// TIA Portal project "TestingMurr" (V18)

(* hardware
DEVICE "S7-1200 station_1"  S7-1200 Station
   slot 0: "Rack_0"  S7-1200 Rack  Rack  V1.0
   slot 1: "PLC_1"  CPU 1212FC DC/DC/DC  6ES7 212-1AF40-0XB0  V4.6
DEVICE "GSD device_1"  GSD.Device.PN
   slot 0: "Rack"  Rack  V1.0
   slot 0: "IMPACT67-Pro"  54630 IMPACT67 Pro PNIO DIO8 IOL8 M12L 5P  54630  V1.5.0
      slot 0: "54630 IMPACT67 Pro PNIO DIO8 IOL8 M12L 5P_1"  54630 IMPACT67 Pro PNIO DIO8 IOL8 M12L 5P
      slot 1: "54630 IMPACT67 Pro PNIO DIO8 IOL8 M12L 5P"  54630 IMPACT67 Pro PNIO DIO8 IOL8 M12L 5P
         slot 1: "Port 1"  Port 1
         slot 2: "Port 2"  Port 2
      slot 1: "IMPACT67 Pro device_1"  IMPACT67 Pro device
         slot 0: "SIO data / Module parameters"  SIO data / Module parameters
      slot 2: "IMPACT67 Pro options_1"  IMPACT67 Pro options
   slot 1: "PortX0-59719 MVP12-P6 DIO16 8xM12A IOLA12 B0"  59719 MVP12-P6 DIO16 8xM12A IOLA12 B0
   slot 2: "Standard digital input"  Standard digital input
   slot 3: "Deactivated_1"  Deactivated
   slot 4: "PortX3-500x-00501-1300001 IOL AI-U/I-STR-MULT-PAR"  500x-00501-1300001 IOL AI-U/I-STR-MULT-PAR
   slot 5: "PortX4-Contrinex _IDWE-M12MM-NMS-A0"  IO-Link In/Out 04/02 bytes + PQI
   slot 6: "Web server"  Web server
   slot 6: "Standard digital output"  Standard digital output
   slot 7: "PortX6-OMRON_E3AS_HL500LMN"  IO-Link In/Out 04/02 bytes + PQI
   slot 8: "PortX7-TURCK_BN1F360V_QR20-IOLX3-H1141"  IO-Link In/Out 08/02 bytes + PQI
*)

// ===== PLC "PLC_1"  CPU 1212FC DC/DC/DC =====

VAR_GLOBAL   // PLC tag table "Default tag table"
   "iwMurrIOLINKData_SIO_IN" AT %I100.0 : "DUT_Murr_Submodule 1_SIO_PortBase_Pin";
   "iwMurrIOLINKData_X4_IN" AT %I114.0 : "DUT_RawArray_Length4";   // PortX4-Contrinex _IDWE-M12MM-NMS-A0
   "iwMurrIOLINKData_X6_IN" AT %I120.0 : "DUT_RawArray_Length4";   // PortX6-OMRON_E3AS_HL500LMN
   "iwMurrIOLINKData_X3_IN" AT %I110.0 : "DUT_RawArray_Length2";   // PortX3-500x-00501-1300001 IOL AI-U/I-STR-MULT-PAR
   "iwMurrIOLINKData_X3_IN_PQI" AT %IB112 : Byte;
   "iwMurrIOLINKData_X4_IN_PQI" AT %IB118 : Byte;
   "iwMurrIOLINKData_IN_X6_PQI" AT %IB124 : Byte;
   "iwMurrIOLINKData_X0_IN" AT %I102.0 : "DUT_RawArray_Length4";   // PortX0-59719 MVP12-P6 DIO16 8xM12A IOLA12 B0
   "iwMurrIOLINKData_X7_IN" AT %I126.0 : "DUT_RawArray_Length8";   // PortX7-TURCK_BN1F360V_QR20-IOLX3-H1141
   "iwMurrIOLINKData_X7_IN_PQI" AT %IB134 : Byte;
   "iwMurrIOLINKData_X0_OUT" AT %Q102.0 : "DUT_RawArray_Length2";
   "iwMurrIOLINKData_SIO_OUT" AT %Q100.0 : "DUT_Murr_Submodule 1_SIO_PortBase_Pin";
   "iwMurrIOLINKData_X5_IN_PQI" AT %IB138 : Byte;   // PortX7-TURCK_BN1F360V_QR20-IOLX3-H1141
   "System_Byte" AT %MB1 : Byte;
   "FirstScan" AT %M1.0 : Bool;
   "DiagStatusUpdate" AT %M1.1 : Bool;
   "AlwaysTRUE" AT %M1.2 : Bool;
   "AlwaysFALSE" AT %M1.3 : Bool;
   "Clock_Byte" AT %MB0 : Byte;
   "Clock_10Hz" AT %M0.0 : Bool;
   "Clock_5Hz" AT %M0.1 : Bool;
   "Clock_2.5Hz" AT %M0.2 : Bool;
   "Clock_2Hz" AT %M0.3 : Bool;
   "Clock_1.25Hz" AT %M0.4 : Bool;
   "Clock_1Hz" AT %M0.5 : Bool;
   "Clock_0.625Hz" AT %M0.6 : Bool;
   "Clock_0.5Hz" AT %M0.7 : Bool;
END_VAR

TYPE "DUT_Murr_Submodule 1_SIO_PortBase_Pin"
   STRUCT
      PortX0Pin4 : Bool;
      PortX0Pin2 : Bool;
      PortX1Pin4 : Bool;
      PortX1Pin2 : Bool;
      PortX2Pin4 : Bool;
      PortX2Pin2 : Bool;
      PortX3Pin4 : Bool;
      PortX3Pin2 : Bool;
      PortX4Pin4 : Bool := false;
      PortX4Pin2 : Bool := false;
      PortX5Pin4 : Bool := false;
      PortX5Pin2 : Bool := false;
      PortX6Pin4 : Bool := false;
      PortX6Pin2 : Bool := false;
      PortX7Pin4 : Bool := false;
      PortX7Pin2 : Bool := false;
   END_STRUCT;
END_TYPE

TYPE "DUT_OMRON_E3AS_HL5000LMN_IN"
   STRUCT
      DetectValueOutput : Int;
      LightIntensityLevel : USInt;
      Status : "DUT_OMRON_E3AS_HL5000LMN_IN_Status";
   END_STRUCT;
END_TYPE

TYPE "DUT_TURCK_BN1F360V_QR20_IOLX3-H1141_IN"
   STRUCT
      InversProcessData : Int;
      ProcessData : Int;
      Scale : SInt;
      VendorSpecific : USInt;
   END_STRUCT;
END_TYPE

TYPE "DUT_TURCK_BN1F360V_QR20_IOLX3-H1141_OUT"
   STRUCT
      ProcessDataOutput : USInt;   // Trigger center point teach function,0-3
   END_STRUCT;
END_TYPE

TYPE "DUT_Contrinex _IDWE_M12MM-NMS_A0_IN_Byte0"
   STRUCT
      OSS1 : Bool;
      OSS2 : Bool;
      TSS : Bool;
      SSC1 : Bool;
      SSC2 : Bool;
      ALR1 : Bool;
      ALR2 : Bool;
      ALR3 : Bool;
   END_STRUCT;
END_TYPE

TYPE "DUT_RawArray_Length4"
   STRUCT
      raw : Array[0..3] of Byte;
   END_STRUCT;
END_TYPE

TYPE "DUT_RawArray_Length8"
   STRUCT
      raw : Array[0..7] of Byte;
   END_STRUCT;
END_TYPE

TYPE "DUT_OMRON_E3AS_HL5000LMN_IN_Status"
   STRUCT
      ControlOutput1 : Bool;
      ControlOutput2 : Bool;
      InstabilityAlarm : Bool;
      InsufficinetError : Bool;
      Warning : Bool;
      Error : Bool;
   END_STRUCT;
END_TYPE

TYPE "DUT_EUROSwitch_LevelSeneor"
   STRUCT
      AnalogData : Real;
      Level : Real;
   END_STRUCT;
END_TYPE

TYPE "DUT_Contrinex _IDWE_M12MM-NMS_A0"
   STRUCT
      Stauts : "DUT_Contrinex _IDWE_M12MM-NMS_A0_IN_Byte0";
      ScaleValue : USInt;
      MeasureValue : Int;
   END_STRUCT;
END_TYPE

TYPE "DUT_Murr_IOLinkMaster_PQI"
   STRUCT
      b0 : Bool;   // Reserved(“0”)
      b1 : Bool;   // Reserved(“0”)
      NewPar : Bool;   // 0=No update of the device parameters detected
      SubstDev : Bool;   // 0=No replacement device detected (identical serial number).
      PortActive : Bool;   // 0=Port disabled via port function.
      DevCom : Bool;   // 0=No device available.
      DevErr : Bool;   // 0=No error/warning occurred.
      PQ : Bool;   // 0=Invalid IO process data from the device.
   END_STRUCT;
END_TYPE

TYPE "DUT_RawArray_Length2"
   STRUCT
      raw : Array[0..1] of Byte;
   END_STRUCT;
END_TYPE

TYPE "DUT_Murr_IOLINKHUB_59719_IN_Bytes2_3"
   STRUCT
      ErrorAtPowerSupply : Bool;   // Power Suppluy Too low/Too High
      ErrorAtTempature : Bool;   // Tempature Over Range
      ErrorAtInOut : Bool;   // Short Circut/Overload
      DIA : SInt;
      GlobalStatus : Bool;   // 0=no diagnostic
      DeviceIdentification : SInt;   // User defined bits
   END_STRUCT;
END_TYPE

TYPE "DUT_Murr_IOLINKHUB_59719_IN"
   STRUCT
      Pin : "DUT_Murr_Submodule 1_SIO_PortBase_Pin";
      Status : "DUT_Murr_IOLINKHUB_59719_IN_Bytes2_3";
   END_STRUCT;
END_TYPE

DATA_BLOCK "Main_Safety_RTG1_DB"   // DB1, F_DB
{ S7_Optimized_Access := 'TRUE' }
NAME : FUSI
VERSION : 0.1
// stored: InstanceOfName Main_Safety_RTG1
"Main_Safety_RTG1"
BEGIN
END_DATA_BLOCK

// folder: DB

DATA_BLOCK "FB_Murr_DB"   // DB2
{ S7_Optimized_Access := 'TRUE' }
VERSION : 0.1
// stored: InstanceOfName FB_Murr
"FB_Murr"
BEGIN
END_DATA_BLOCK

DATA_BLOCK "DB_MurrIOLINK_Data"   // DB3
{ S7_Optimized_Access := 'TRUE' }
VERSION : 0.1
   VAR
      X0 : Struct
         IOLinkIN : "DUT_Murr_IOLINKHUB_59719_IN";
         IOLinkOUT : "DUT_Murr_Submodule 1_SIO_PortBase_Pin";
      END_STRUCT;
      X3 : Struct
         IOLinkIN : "DUT_EUROSwitch_LevelSeneor";
         PQI : "DUT_Murr_IOLinkMaster_PQI";
      END_STRUCT;
      X4 : Struct
         IOLinkIN : "DUT_Contrinex _IDWE_M12MM-NMS_A0";
         PQI : "DUT_Murr_IOLinkMaster_PQI";
      END_STRUCT;
      X6 : Struct
         IOLinkIN : "DUT_OMRON_E3AS_HL5000LMN_IN";
         PQI : "DUT_Murr_IOLinkMaster_PQI";
      END_STRUCT;
      X7 : Struct
         IOLinkIN : "DUT_TURCK_BN1F360V_QR20_IOLX3-H1141_IN";
         PQI : "DUT_Murr_IOLinkMaster_PQI";
      END_STRUCT;
   END_VAR
BEGIN
END_DATA_BLOCK

// folder: (top level)

FUNCTION_BLOCK "Main_Safety_RTG1"   // FB1, F_FBD
{ S7_Optimized_Access := 'TRUE' }
BEGIN
END_FUNCTION_BLOCK

ORGANIZATION_BLOCK "Main"   // OB1, LAD, ProgramCycle
TITLE = "Main Program Sweep (Cycle)"
{ S7_Optimized_Access := 'TRUE' }
VERSION : 0.1
   VAR_INPUT
      Initial_Call : Bool;   // Initial call of this OB
      Remanence : Bool;   // =True, if remanent data are available
   END_VAR
BEGIN

REGION Network 2
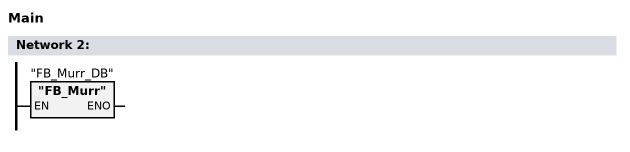
   RUNG wire#powerrail
      "FB_Murr_DB"()
   END_RUNG
   // the same network as SCL:
   "FB_Murr_DB"();   // "FB_Murr"
END_REGION
END_ORGANIZATION_BLOCK

// folder: FB

FUNCTION_BLOCK "FB_Murr"   // FB3, FBD
{ S7_Optimized_Access := 'TRUE' }
VERSION : 0.1
   VAR
      X0 : "FB_Murr_IOLINKHUB_59719";
      X4 : "FB_Contrinex _IDWE_M12MM-NMS_A0";
      X5 : "FB_EUROSwitch_LevelSeneor";
      X6 : "FB_OMRON_E3AS_HL5000LMN";
      X7 : "FB_TURCK_BN1F360V_QR20_IOLX3_H1141";
      PQIs : Array[0..7] of "FB_Murr_IOLINKDevices_PQI";
   END_VAR
BEGIN

REGION Network 1: SIO
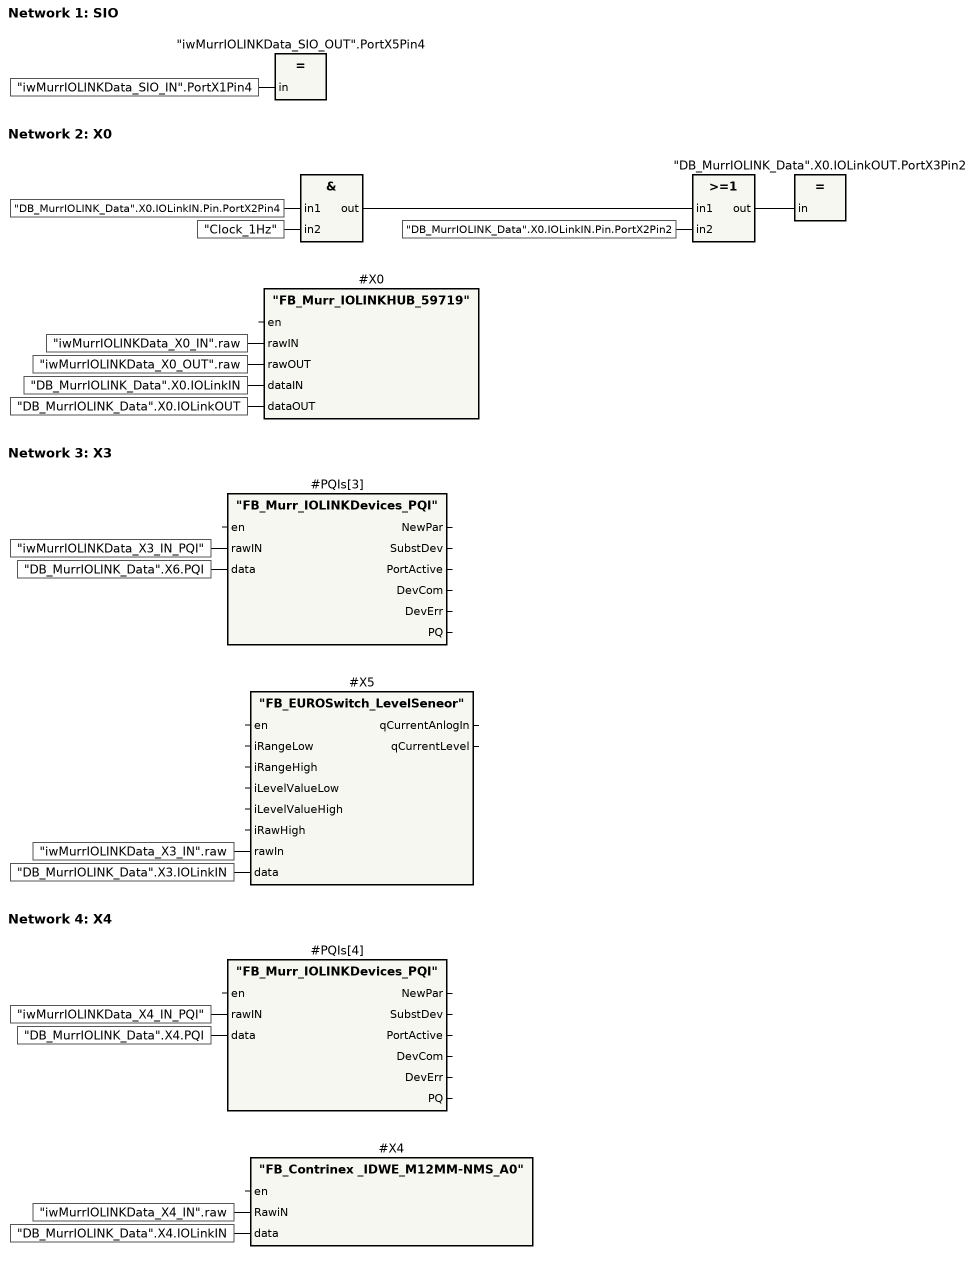
   "iwMurrIOLINKData_SIO_OUT".PortX5Pin4 := "iwMurrIOLINKData_SIO_IN".PortX1Pin4;
END_REGION

REGION Network 2: X0
   "DB_MurrIOLINK_Data".X0.IOLinkOUT.PortX3Pin2 := ("DB_MurrIOLINK_Data".X0.IOLinkIN.Pin.PortX2Pin4 AND "Clock_1Hz") OR "DB_MurrIOLINK_Data".X0.IOLinkIN.Pin.PortX2Pin2;
   #X0(rawIN := "iwMurrIOLINKData_X0_IN".raw,   // "FB_Murr_IOLINKHUB_59719"
       rawOUT := "iwMurrIOLINKData_X0_OUT".raw,
       dataIN := "DB_MurrIOLINK_Data".X0.IOLinkIN,
       dataOUT := "DB_MurrIOLINK_Data".X0.IOLinkOUT);
END_REGION

REGION Network 3: X3
   #PQIs[3](rawIN := "iwMurrIOLINKData_X3_IN_PQI", data := "DB_MurrIOLINK_Data".X6.PQI);   // "FB_Murr_IOLINKDevices_PQI"
   #X5(rawIn := "iwMurrIOLINKData_X3_IN".raw, data := "DB_MurrIOLINK_Data".X3.IOLinkIN);   // "FB_EUROSwitch_LevelSeneor"
END_REGION

REGION Network 4: X4
   #PQIs[4](rawIN := "iwMurrIOLINKData_X4_IN_PQI", data := "DB_MurrIOLINK_Data".X4.PQI);   // "FB_Murr_IOLINKDevices_PQI"
   #X4(RawiN := "iwMurrIOLINKData_X4_IN".raw, data := "DB_MurrIOLINK_Data".X4.IOLinkIN);   // "FB_Contrinex _IDWE_M12MM-NMS_A0"
END_REGION

REGION Network 5: X6
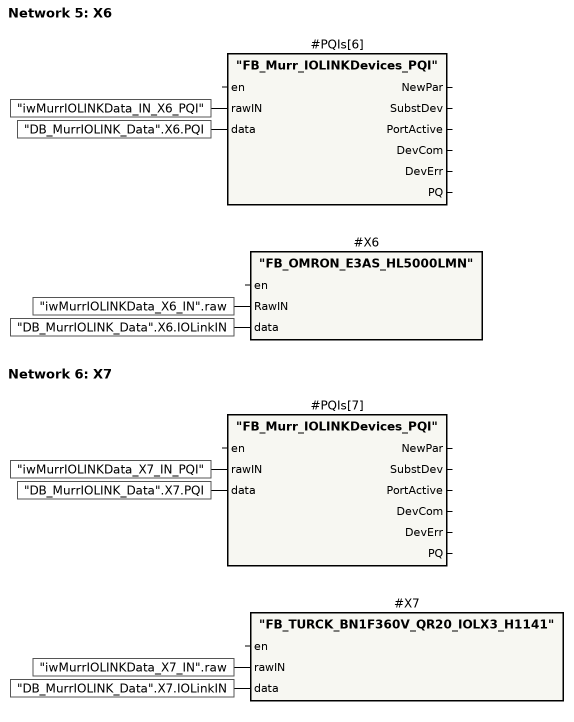
   #PQIs[6](rawIN := "iwMurrIOLINKData_IN_X6_PQI", data := "DB_MurrIOLINK_Data".X6.PQI);   // "FB_Murr_IOLINKDevices_PQI"
   #X6(RawIN := "iwMurrIOLINKData_X6_IN".raw, data := "DB_MurrIOLINK_Data".X6.IOLinkIN);   // "FB_OMRON_E3AS_HL5000LMN"
END_REGION

REGION Network 6: X7
   #PQIs[7](rawIN := "iwMurrIOLINKData_X7_IN_PQI", data := "DB_MurrIOLINK_Data".X7.PQI);   // "FB_Murr_IOLINKDevices_PQI"
   #X7(rawIN := "iwMurrIOLINKData_X7_IN".raw, data := "DB_MurrIOLINK_Data".X7.IOLinkIN);   // "FB_TURCK_BN1F360V_QR20_IOLX3_H1141"
END_REGION
END_FUNCTION_BLOCK

// folder: FB/FB_Sensors

FUNCTION_BLOCK "FB_Contrinex _IDWE_M12MM-NMS_A0"   // FB2, FBD
{ S7_Optimized_Access := 'TRUE' }
VERSION : 0.1
   VAR_IN_OUT
      RawiN : Array[0..3] of Byte;
      data : "DUT_Contrinex _IDWE_M12MM-NMS_A0";
   END_VAR
   VAR_TEMP
      pos : DInt;
      ReVal : Word;
   END_VAR
BEGIN

REGION Network 1: OSS1
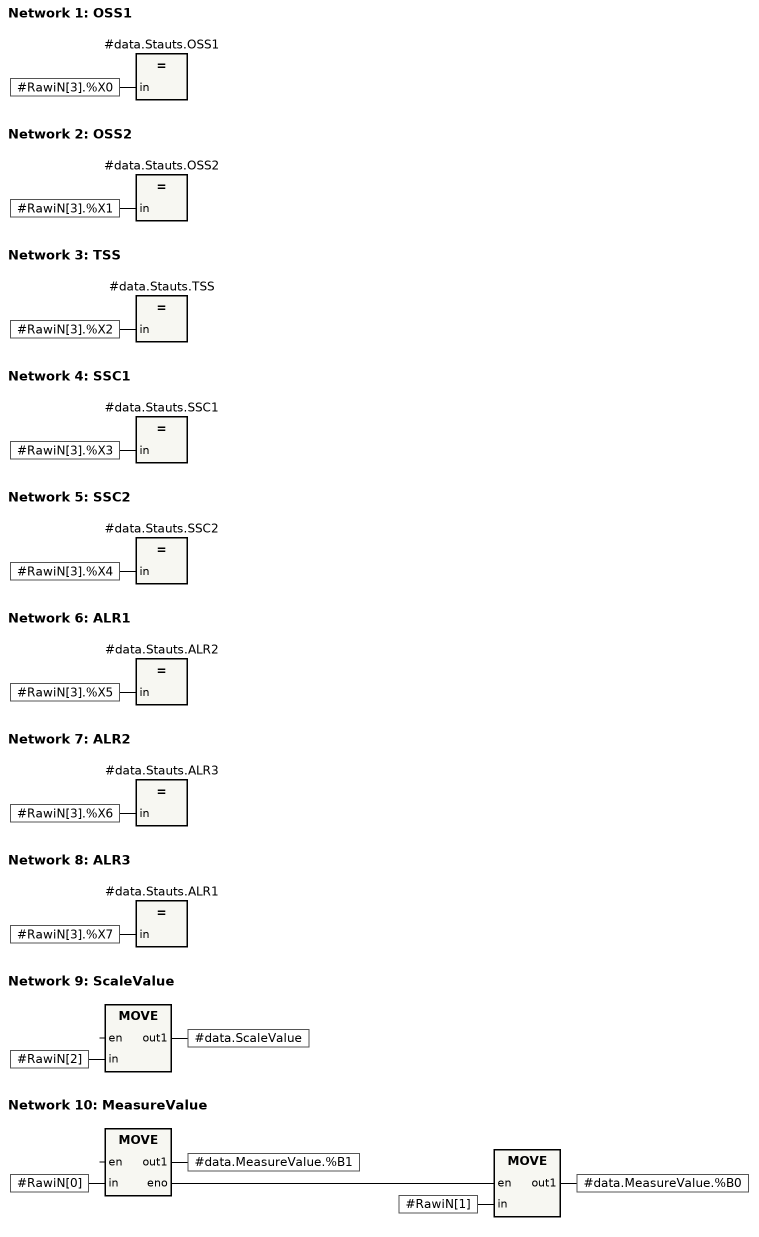
   #data.Stauts.OSS1 := #RawiN[3].%X0;
END_REGION

REGION Network 2: OSS2
   #data.Stauts.OSS2 := #RawiN[3].%X1;
END_REGION

REGION Network 3: TSS
   #data.Stauts.TSS := #RawiN[3].%X2;
END_REGION

REGION Network 4: SSC1
   #data.Stauts.SSC1 := #RawiN[3].%X3;
END_REGION

REGION Network 5: SSC2
   #data.Stauts.SSC2 := #RawiN[3].%X4;
END_REGION

REGION Network 6: ALR1
   #data.Stauts.ALR2 := #RawiN[3].%X5;
END_REGION

REGION Network 7: ALR2
   #data.Stauts.ALR3 := #RawiN[3].%X6;
END_REGION

REGION Network 8: ALR3
   #data.Stauts.ALR1 := #RawiN[3].%X7;
END_REGION

REGION Network 9: ScaleValue
   #data.ScaleValue := #RawiN[2];
END_REGION

REGION Network 10: MeasureValue
   #data.MeasureValue.%B1 := #RawiN[0];
   #data.MeasureValue.%B0 := #RawiN[1];
END_REGION
END_FUNCTION_BLOCK

FUNCTION_BLOCK "FB_OMRON_E3AS_HL5000LMN"   // FB4, FBD
{ S7_Optimized_Access := 'TRUE' }
VERSION : 0.1
   VAR_IN_OUT
      RawIN : Array[0..3] of Byte;
      data : "DUT_OMRON_E3AS_HL5000LMN_IN";
   END_VAR
BEGIN

REGION Network 1
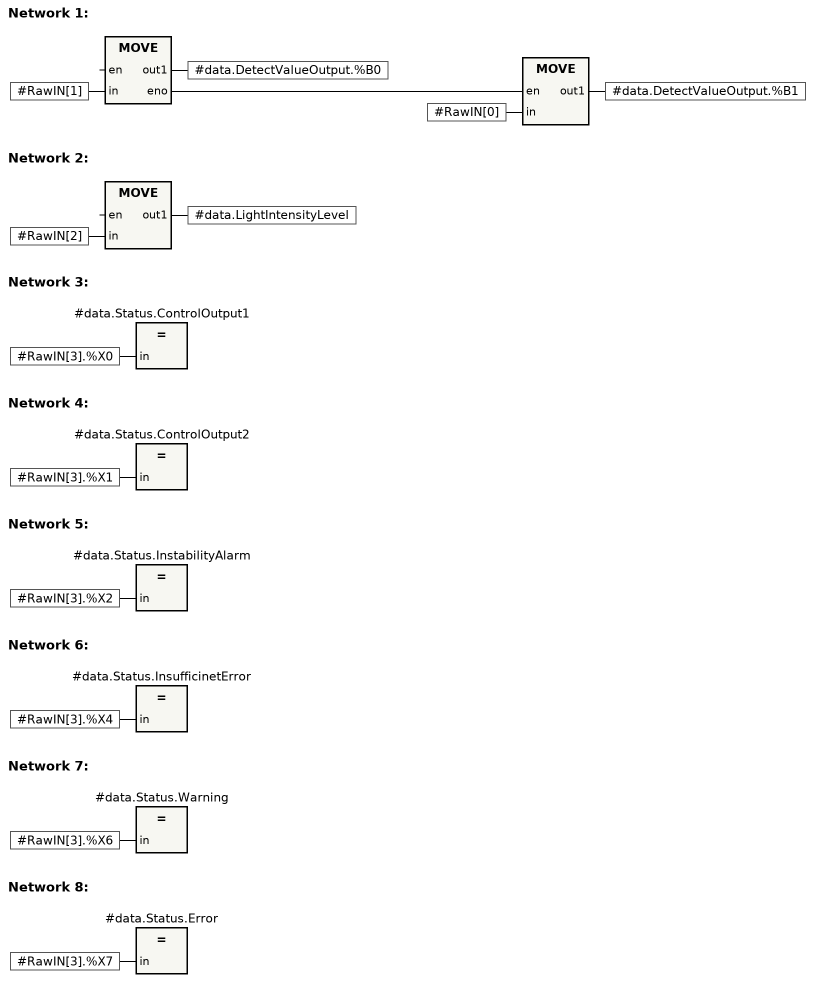
   #data.DetectValueOutput.%B0 := #RawIN[1];
   #data.DetectValueOutput.%B1 := #RawIN[0];
END_REGION

REGION Network 2
   #data.LightIntensityLevel := #RawIN[2];
END_REGION

REGION Network 3
   #data.Status.ControlOutput1 := #RawIN[3].%X0;
END_REGION

REGION Network 4
   #data.Status.ControlOutput2 := #RawIN[3].%X1;
END_REGION

REGION Network 5
   #data.Status.InstabilityAlarm := #RawIN[3].%X2;
END_REGION

REGION Network 6
   #data.Status.InsufficinetError := #RawIN[3].%X4;
END_REGION

REGION Network 7
   #data.Status.Warning := #RawIN[3].%X6;
END_REGION

REGION Network 8
   #data.Status.Error := #RawIN[3].%X7;
END_REGION
END_FUNCTION_BLOCK

FUNCTION_BLOCK "FB_EUROSwitch_LevelSeneor"   // FB5, FBD
{ S7_Optimized_Access := 'TRUE' }
VERSION : 0.1
   VAR_INPUT
      iRangeLow : Real := 4.0;
      iRangeHigh : Real := 20.0;
      iLevelValueLow : Real := 0.0;
      iLevelValueHigh : Real := 100.0;
      iRawHigh : Real := 27676.0;
   END_VAR
   VAR_OUTPUT
      qCurrentAnlogIn : Real;
      qCurrentLevel : Real;
   END_VAR
   VAR_IN_OUT
      rawIn : Array[0..1] of Byte;
      data : "DUT_EUROSwitch_LevelSeneor";
   END_VAR
   VAR
      _INT : Int;
      _real : Real;
   END_VAR
BEGIN

REGION Network 1
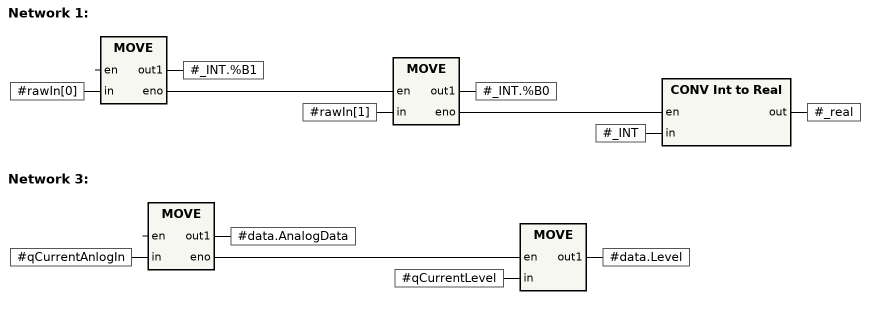
   #_INT.%B1 := #rawIn[0];
   #_INT.%B0 := #rawIn[1];
   #_real := INT_TO_REAL(#_INT);
END_REGION

REGION Network 2 (SCL)
   #qCurrentAnlogIn :=
   (#_real / #iRawHigh) * #iRangeHigh + #iRangeLow;

   #qCurrentLevel :=
   (#_real / #iRawHigh) * #iLevelValueHigh + #iLevelValueLow;
END_REGION

REGION Network 3
   #data.AnalogData := #qCurrentAnlogIn;
   #data.Level := #qCurrentLevel;
END_REGION
END_FUNCTION_BLOCK

FUNCTION_BLOCK "FB_Murr_IOLINKDevices_PQI"   // FB6, FBD
{ S7_Optimized_Access := 'TRUE' }
VERSION : 0.1
   VAR_OUTPUT
      NewPar : Bool;   // 0=No update of the device parameters detected
      SubstDev : Bool;   // 0=No replacement device detected (identical serial number).
      PortActive : Bool;   // 0=Port disabled via port function.
      DevCom : Bool;   // 0=No device available.
      DevErr : Bool;   // 0=No error/warning occurred.
      PQ : Bool;   // 0=Invalid IO process data from the device.
   END_VAR
   VAR_IN_OUT
      rawIN : Byte;
      data : "DUT_Murr_IOLinkMaster_PQI";
   END_VAR
BEGIN

REGION Network 1
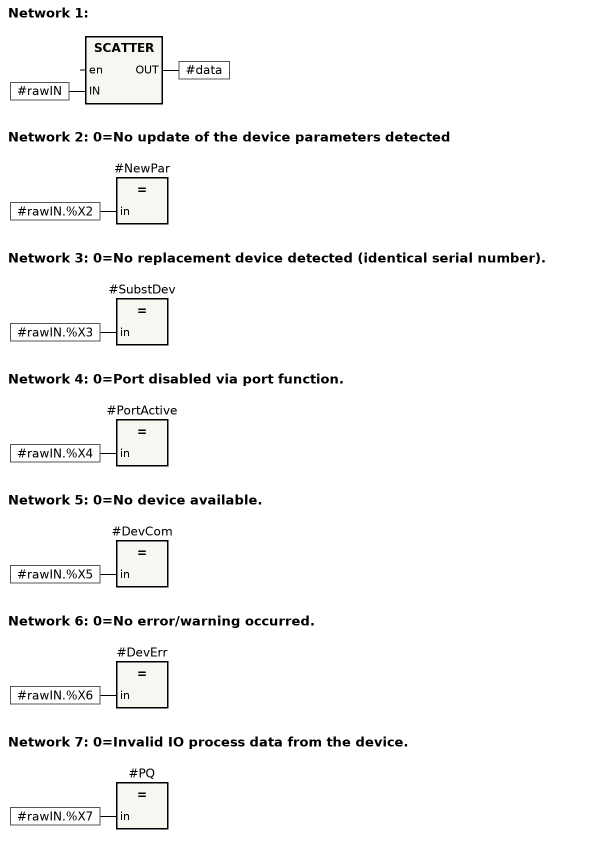
   SCATTER(IN := #rawIN, OUT => #data);
END_REGION

REGION Network 2: 0=No update of the device parameters detected
   #NewPar := #rawIN.%X2;
END_REGION

REGION Network 3: 0=No replacement device detected (identical serial number).
   #SubstDev := #rawIN.%X3;
END_REGION

REGION Network 4: 0=Port disabled via port function.
   #PortActive := #rawIN.%X4;
END_REGION

REGION Network 5: 0=No device available.
   #DevCom := #rawIN.%X5;
END_REGION

REGION Network 6: 0=No error/warning occurred.
   #DevErr := #rawIN.%X6;
END_REGION

REGION Network 7: 0=Invalid IO process data from the device.
   #PQ := #rawIN.%X7;
END_REGION
END_FUNCTION_BLOCK

FUNCTION_BLOCK "FB_Murr_IOLINKHUB_59719"   // FB7, FBD
{ S7_Optimized_Access := 'TRUE' }
VERSION : 0.1
   VAR_IN_OUT
      rawIN : Array[*] of Byte;
      rawOUT : Array[*] of Byte;
      dataIN : "DUT_Murr_IOLINKHUB_59719_IN";
      dataOUT : "DUT_Murr_Submodule 1_SIO_PortBase_Pin";
   END_VAR
   VAR_TEMP
      _word : Word;
   END_VAR
BEGIN

REGION Network 1
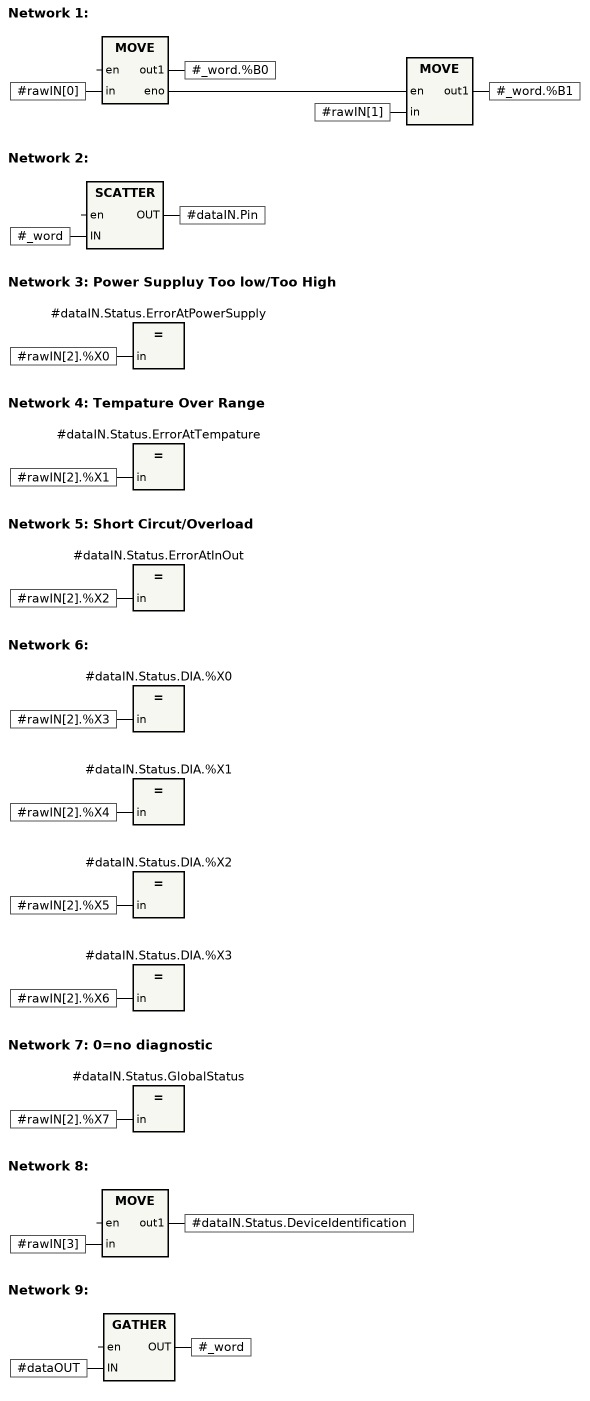
   #_word.%B0 := #rawIN[0];
   #_word.%B1 := #rawIN[1];
END_REGION

REGION Network 2
   SCATTER(IN := #_word, OUT => #dataIN.Pin);
END_REGION

REGION Network 3: Power Suppluy Too low/Too High
   #dataIN.Status.ErrorAtPowerSupply := #rawIN[2].%X0;
END_REGION

REGION Network 4: Tempature Over Range
   #dataIN.Status.ErrorAtTempature := #rawIN[2].%X1;
END_REGION

REGION Network 5: Short Circut/Overload
   #dataIN.Status.ErrorAtInOut := #rawIN[2].%X2;
END_REGION

REGION Network 6
   #dataIN.Status.DIA.%X0 := #rawIN[2].%X3;
   #dataIN.Status.DIA.%X1 := #rawIN[2].%X4;
   #dataIN.Status.DIA.%X2 := #rawIN[2].%X5;
   #dataIN.Status.DIA.%X3 := #rawIN[2].%X6;
END_REGION

REGION Network 7: 0=no diagnostic
   #dataIN.Status.GlobalStatus := #rawIN[2].%X7;
END_REGION

REGION Network 8
   #dataIN.Status.DeviceIdentification := #rawIN[3];
END_REGION

REGION Network 9
   GATHER(IN := #dataOUT, OUT => #_word);
END_REGION

REGION Network 10
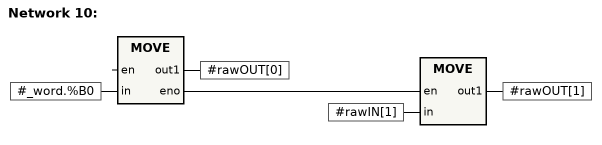
   #rawOUT[0] := #_word.%B0;
   #rawOUT[1] := #rawIN[1];
END_REGION
END_FUNCTION_BLOCK

FUNCTION_BLOCK "FB_TURCK_BN1F360V_QR20_IOLX3_H1141"   // FB8, FBD
{ S7_Optimized_Access := 'TRUE' }
VERSION : 0.1
   VAR_IN_OUT
      rawIN : Array[*] of Byte;
      data : "DUT_TURCK_BN1F360V_QR20_IOLX3-H1141_IN";
   END_VAR
   VAR_TEMP
      _word : Word;
   END_VAR
BEGIN

REGION Network 1
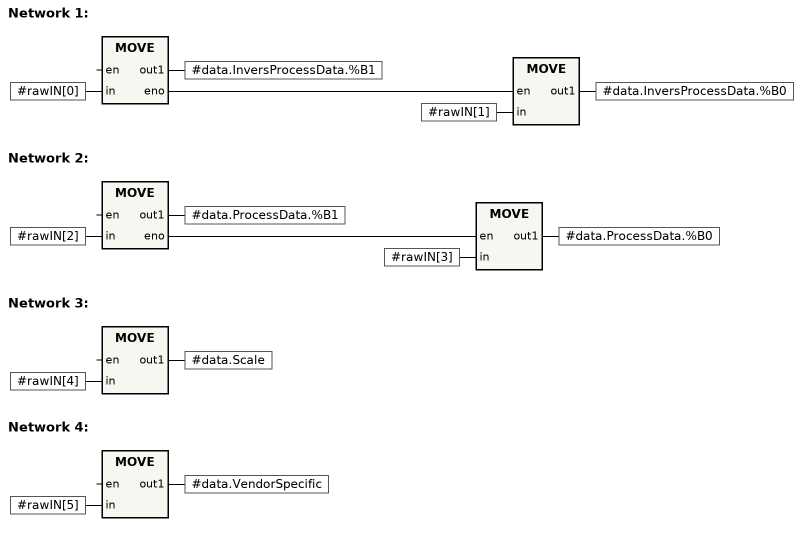
   #data.InversProcessData.%B1 := #rawIN[0];
   #data.InversProcessData.%B0 := #rawIN[1];
END_REGION

REGION Network 2
   #data.ProcessData.%B1 := #rawIN[2];
   #data.ProcessData.%B0 := #rawIN[3];
END_REGION

REGION Network 3
   #data.Scale := #rawIN[4];
END_REGION

REGION Network 4
   #data.VendorSpecific := #rawIN[5];
END_REGION
END_FUNCTION_BLOCK